// TwinCAT 3 PLC project DemoPLC
// ProgramVersion: 3.1.4026.22
// libraries:
//   Tc2_MC2, * (Beckhoff Automation GmbH)
//   Tc2_MDP, * (Beckhoff Automation GmbH)
//   Tc2_Standard, * (Beckhoff Automation GmbH)
//   Tc2_System, * (Beckhoff Automation GmbH)
//   Tc2_Utilities, * (Beckhoff Automation GmbH)
//   Tc3_IPCDiag, * (Beckhoff Automation GmbH)
// project tree:
//   DUTs/Bleutooth/ ST_Bleutooth.TcDUT, ST_BleutoothControl.TcDUT, ST_Bleutooth_Status.TcDUT
//   DUTs/CPU/ ST_CPUData.TcDUT, ST_CPUTemperature.TcDUT, ST_CPUUsage.TcDUT, ST_TaskData.TcDUT
//   DUTs/EtherCATJunction/ ST_MS4208_ETCOut.TcDUT
//   DUTs/General/ ST_EFU_Data.TcDUT, ST_EFU_Device_Inputs.TcDUT, ST_EFU_Inputs.TcDUT, ST_EFU_Outputs.TcDUT
//   DUTs/IO/DCombi/ ST_MO2338_DCombi.TcDUT
//   DUTs/IO/DI/ ST_DIS_Chanel_Diagnosis.TcDUT, ST_DIS_Diagnosis.TcDUT, ST_DIS_Inputs.TcDUT, ST_MO1008_DI.TcDUT
//   DUTs/IO/DO/ ST_DOS_Diagnosis.TcDUT, ST_DOS_Output.TcDUT, ST_DOS_Chanel_Diagnosis.TcDUT, ST_MO2008_DO.TcDUT
//   DUTs/PSU/ ST_PSU_Data.TcDUT, ST_PSU_Inputs.TcDUT, ST_PSU_Outputs.TcDUT
//   GVLs/ Global_Managed_Variables.TcGVL
//   / PlcTask.TcTTO
//   POUs/ FB_CollectCPUData.TcPOU, MAIN.TcPOU
//   POUs/Motion/Duts/ E_DemoSteps.TcTLEO, ST_PositionParameters.TcDUT
//   POUs/Motion/ FB_DemoMotion.TcPOU
//   POUs/Utilities/ FB_Blink.TcPOU
// real-time tasks:
//   TASK PlcTask: cycle T#10ms, priority 20, ADS port 350
// motion (NC):
//   TASK NC-Task 1 SAF: cycle T#2ms, priority 4, ADS port 501
//   TASK NC-Task 1 SVB: cycle T#10ms, priority 8, ADS port 511
//   AXIS Axis 2 (id 2)
//     General: UnitName=°
//     Dynamic: Acceleration=15000, Deceleration=15000, Jerk=118292.94
//     Velo: RefSearch=262.8732, RefSync=262.8732, SlowManual=1314.366, FastManual=7886.196, Fast=26287.32, Maximum=26287.32
//     OtherSettings: AllowMotionCmdToSlave=true
//     encoder EncType=19
//       EncPara: ScaleFactorNumerator=360, ScaleFactorDenominator=1048576, MaxCount=#xffffffff
//     drive DrvType=16
//       DrvPara: MaxCount=#xffffffff, DriveControlDWord=#x00020100
//         Analog: VeloReferenz=28916.052, VeloScale=32, TorqueSetpointScale=10, ScaleFactorActTorque=0.1
//         TimeComp: TaskDelayCycles=1
//     controller CtrType=1
//       CtrPara: PriorControlFactor=1
//         PID: PosKp=5
//         Observer: BandWidth=20
// I/O:
//   DEVICE Device 1 (EtherCAT), AmsNetId 10.201.45.9.2.1
//     Term 14 (MB1200-0000)
// variable links:
//   (this object) <-> Device 1 (EtherCAT)/Term 14 (MB1200-0000)/Term 8 (MB1100-0002)/Term 11 (MO7221-9016-1114)
//     Drive/Inputs/In/nDataIn1 <-> DRV Following error actual value/Following error actual value
//     Drive/Inputs/In/nDataIn3[0] <-> DRV Torque actual value/Torque actual value
//     Drive/Inputs/In/nDcOutputTime <-> InfoData/DcOutputShift
//     Drive/Inputs/In/nState1 <-> DRV Statusword/Statusword
//     Drive/Inputs/In/nState2 <-> DRV Statusword/Statusword @bit 8
//     Drive/Inputs/In/nState4 @bit 1 <-> WcState/InputToggle0
//     Drive/Inputs/In/nState4 <-> WcState/WcState0
//     Drive/Outputs/Out/nCtrl1 <-> DRV Controlword/Controlword
//     Drive/Outputs/Out/nCtrl2 <-> DRV Controlword/Controlword @bit 8
//     Drive/Outputs/Out/nDataOut1 <-> DRV Target position/Target position
//     Enc/Inputs/In/nDataIn1 <-> FB Position/Position
//     Enc/Inputs/In/nDcInputTime <-> InfoData/DcInputShift
//     Enc/Inputs/In/nState2 @bit 6 <-> FB Status/Status/Input cycle counter
//     Enc/Inputs/In/nState2 @bit 5 <-> FB Status/Status/TxPDO State
//     Enc/Inputs/In/nState4 @bit 1 <-> WcState/InputToggle0
//     Enc/Inputs/In/nState4 <-> WcState/WcState0
//     PlcTask Inputs/MAIN.fbDemoMotion.bSafety_Error <-> Module 1 (SafetyMDSingle)/Standard Inputdata/Standard Out Var 9
//     PlcTask Inputs/MAIN.fbDemoMotion.bSafety_OK <-> Module 1 (SafetyMDSingle)/Standard Inputdata/Standard Out Var 8
//     PlcTask Outputs/MAIN.bRunSafety <-> Module 1 (SafetyMDSingle)/Standard Outputdata/Standard In Var 2
//     PlcTask Outputs/MAIN.fbDemoMotion.bSafety_ErrorAckFromPLC <-> Module 1 (SafetyMDSingle)/Standard Outputdata/Standard In Var 1
//     PlcTask Outputs/MAIN.fbDemoMotion.bSafety_ErrorAckFromPLC <-> Module 1 (SafetyMDSingle)/Standard Outputdata/Standard In Var 7
//     PlcTask Outputs/MAIN.fbDemoMotion.bSafety_STOFromPLC <-> Module 1 (SafetyMDSingle)/Standard Outputdata/Standard In Var 6
//   (this object) <-> Device 1 (EtherCAT)/Term 14 (MB1200-0000)/Term 8 (MB1100-0002)
//     PlcTask Inputs/MAIN.stBleuToothData.Status/BleutoothEnabled <-> BTG Inputs/Status/Bluetooth Enabled
//     PlcTask Inputs/MAIN.stBleuToothData.Status/Connected <-> BTG Inputs/Status/Connected
//     PlcTask Inputs/MAIN.stBleuToothData.Status/Diag <-> BTG Inputs/Status/Diag
//     PlcTask Inputs/MAIN.stBleuToothData.Status/DonglePresent <-> BTG Inputs/Status/Dongle Present
//     PlcTask Inputs/MAIN.stBleuToothData.Status/Pairing <-> BTG Inputs/Status/Pairing Active
//     PlcTask Outputs/MAIN.stBleuToothData.control/ActivatePairingMode <-> BTG Outputs/Control/Activate Pairing
//     PlcTask Outputs/MAIN.stBleuToothData.control/EnableBleutoothDiagnosis <-> BTG Outputs/Control/Enable Bluetooth
//   (this object) <-> Device 1 (EtherCAT)/Term 14 (MB1200-0000)/Term 8 (MB1100-0002)/Term 16 (MS1010-1002-1334)
//     PlcTask Inputs/MAIN.stPSUData.stPSUInputs/DCOk <-> PSU Inputs/DC OK
//     PlcTask Inputs/MAIN.stPSUData.stPSUInputs/Overrange <-> PSU Inputs/Overrange
//     PlcTask Inputs/MAIN.stPSUData.stPSUInputs/bError <-> PSU Inputs/Error
//     PlcTask Inputs/MAIN.stPSUData.stPSUInputs/bI2TWarning <-> PSU Inputs/I2T Warning
//     PlcTask Inputs/MAIN.stPSUData.stPSUInputs/bWarning <-> PSU Inputs/Warning
//     PlcTask Inputs/MAIN.stPSUData.stPSUInputs/fActualOutputCurrent <-> PSU Inputs/Output Current
//     PlcTask Inputs/MAIN.stPSUData.stPSUInputs/fActualOutputVoltage <-> PSU Inputs/Output Voltage
//     PlcTask Inputs/MAIN.stPSUData.stPSUInputs/nActualI2TUtilization <-> PSU Inputs/I2T Utilization
//     PlcTask Inputs/MAIN.stPSUData.stPSUInputs/nInfoData1 <-> PSU Inputs/Info Data 1
//     PlcTask Inputs/MAIN.stPSUData.stPSUInputs/nInfoData2 <-> PSU Inputs/Info Data 2
//     PlcTask Outputs/MAIN.stPSUData.stPSUOutputs/bDisableOutput <-> PSU Outputs/Disable Output
//     PlcTask Outputs/MAIN.stPSUData.stPSUOutputs/bReset <-> PSU Outputs/Reset
//   (this object) <-> Device 1 (EtherCAT)/Term 14 (MB1200-0000)/Term 8 (MB1100-0002)/Term 18 (MB1120)/Term 19 (MS4208-2003-1112)
//     PlcTask Inputs/MAIN.st_MS4208_EtherCATOut.stEFUInputsDevice/bDiag <-> EFU Device Inputs/Diag
//     PlcTask Inputs/MAIN.st_MS4208_EtherCATOut.stEFUInputsDevice/bError <-> EFU Device Inputs/Error
//     PlcTask Inputs/MAIN.st_MS4208_EtherCATOut.stEFUInputsDevice/bOvertemperatureWarning <-> EFU Device Inputs/Overtemperature Warning
//     PlcTask Inputs/MAIN.st_MS4208_EtherCATOut.stEFUInputsDevice/bUnderVoltage_Up <-> EFU Device Inputs/Undervoltage Up
//     PlcTask Inputs/MAIN.st_MS4208_EtherCATOut.stEFUInputsDevice/bUnderVoltage_Us <-> EFU Device Inputs/Undervoltage Us
//     PlcTask Inputs/MAIN.st_MS4208_EtherCATOut.stEFUInputsDevice/bWarning <-> EFU Device Inputs/Warning
//     PlcTask Inputs/MAIN.st_MS4208_EtherCATOut.stEFUInputsDevice/fTotalCurrent <-> EFU Device Inputs/Total Current
//     PlcTask Inputs/MAIN.st_MS4208_EtherCATOut.stEFUUs.EFUInputs/bEnabled <-> EFU Us Inputs/Enabled
//     PlcTask Inputs/MAIN.st_MS4208_EtherCATOut.stEFUUs.EFUInputs/bError <-> EFU Us Inputs/Error
//     PlcTask Inputs/MAIN.st_MS4208_EtherCATOut.stEFUUs.EFUInputs/bTripped <-> EFU Us Inputs/Tripped
//     PlcTask Inputs/MAIN.st_MS4208_EtherCATOut.stEFUUs.EFUInputs/bWarning <-> EFU Us Inputs/Warning
//     PlcTask Inputs/MAIN.st_MS4208_EtherCATOut.stEFUUs.EFUInputs/fCurrent <-> EFU Us Inputs/Current
//     PlcTask Inputs/MAIN.st_MS4208_EtherCATOut.stEFU_Up1.EFUInputs/bEnabled <-> EFU Up1 Inputs/Enabled
//     PlcTask Inputs/MAIN.st_MS4208_EtherCATOut.stEFU_Up2.EFUInputs/bEnabled <-> EFU Up2 Inputs/Enabled
//     PlcTask Inputs/MAIN.st_MS4208_EtherCATOut.stEFU_Up1.EFUInputs/bError <-> EFU Up1 Inputs/Error
//     PlcTask Inputs/MAIN.st_MS4208_EtherCATOut.stEFU_Up2.EFUInputs/bError <-> EFU Up2 Inputs/Error
//     PlcTask Inputs/MAIN.st_MS4208_EtherCATOut.stEFU_Up1.EFUInputs/bTripped <-> EFU Up1 Inputs/Tripped
//     PlcTask Inputs/MAIN.st_MS4208_EtherCATOut.stEFU_Up2.EFUInputs/bTripped <-> EFU Up2 Inputs/Tripped
//     PlcTask Inputs/MAIN.st_MS4208_EtherCATOut.stEFU_Up1.EFUInputs/bWarning <-> EFU Up1 Inputs/Warning
//     PlcTask Inputs/MAIN.st_MS4208_EtherCATOut.stEFU_Up2.EFUInputs/bWarning <-> EFU Up2 Inputs/Warning
//     PlcTask Inputs/MAIN.st_MS4208_EtherCATOut.stEFU_Up1.EFUInputs/fCurrent <-> EFU Up1 Inputs/Current
//     PlcTask Inputs/MAIN.st_MS4208_EtherCATOut.stEFU_Up2.EFUInputs/fCurrent <-> EFU Up2 Inputs/Current
//     PlcTask Outputs/MAIN.st_MS4208_EtherCATOut.stEFUUs.EFUOutputs/ControlViaProcessData <-> EFU Us Outputs/Control via Process Data
//     PlcTask Outputs/MAIN.st_MS4208_EtherCATOut.stEFUUs.EFUOutputs/bEnable <-> EFU Us Outputs/Enable
//     PlcTask Outputs/MAIN.st_MS4208_EtherCATOut.stEFUUs.EFUOutputs/bReset <-> EFU Us Outputs/Reset
//     PlcTask Outputs/MAIN.st_MS4208_EtherCATOut.stEFU_Up1.EFUOutputs/ControlViaProcessData <-> EFU Up1 Outputs/Control via Process Data
//     PlcTask Outputs/MAIN.st_MS4208_EtherCATOut.stEFU_Up2.EFUOutputs/ControlViaProcessData <-> EFU Up2 Outputs/Control via Process Data
//     PlcTask Outputs/MAIN.st_MS4208_EtherCATOut.stEFU_Up1.EFUOutputs/bEnable <-> EFU Up1 Outputs/Enable
//     PlcTask Outputs/MAIN.st_MS4208_EtherCATOut.stEFU_Up2.EFUOutputs/bEnable <-> EFU Up2 Outputs/Enable
//     PlcTask Outputs/MAIN.st_MS4208_EtherCATOut.stEFU_Up1.EFUOutputs/bReset <-> EFU Up1 Outputs/Reset
//     PlcTask Outputs/MAIN.st_MS4208_EtherCATOut.stEFU_Up2.EFUOutputs/bReset <-> EFU Up2 Outputs/Reset
//   (this object) <-> Device 1 (EtherCAT)/Term 14 (MB1200-0000)/Term 8 (MB1100-0002)/Term 20 (MO1008-0000-1111)
//     PlcTask Inputs/MAIN.St_MO1008_DIData.EFUInputs/bEnabled <-> EFU Inputs/Enabled
//     PlcTask Inputs/MAIN.St_MO1008_DIData.EFUInputs/bError <-> EFU Inputs/Error
//     PlcTask Inputs/MAIN.St_MO1008_DIData.EFUInputs/bTripped <-> EFU Inputs/Tripped
//     PlcTask Inputs/MAIN.St_MO1008_DIData.EFUInputs/bWarning <-> EFU Inputs/Warning
//     PlcTask Inputs/MAIN.St_MO1008_DIData.EFUInputs/fCurrent <-> EFU Inputs/Current
//     PlcTask Outputs/MAIN.St_MO1008_DIData.ModuleDiagnostics.EFUOutputs/ControlViaProcessData <-> EFU Outputs/Control Via Process Data
//     PlcTask Outputs/MAIN.St_MO1008_DIData.ModuleDiagnostics.EFUOutputs/bEnable <-> EFU Outputs/Enable
//     PlcTask Outputs/MAIN.St_MO1008_DIData.ModuleDiagnostics.EFUOutputs/bReset <-> EFU Outputs/Reset
//   (this object) <-> Device 1 (EtherCAT)/Term 14 (MB1200-0000)/Term 8 (MB1100-0002)/Term 23 (MO2008-0000-1111)
//     PlcTask Inputs/MAIN.st_MO2008_DOData.EFUInputs/bEnabled <-> EFU Inputs/Enabled
//     PlcTask Inputs/MAIN.st_MO2008_DOData.EFUInputs/bError <-> EFU Inputs/Error
//     PlcTask Inputs/MAIN.st_MO2008_DOData.EFUInputs/bTripped <-> EFU Inputs/Tripped
//     PlcTask Inputs/MAIN.st_MO2008_DOData.EFUInputs/bWarning <-> EFU Inputs/Warning
//     PlcTask Inputs/MAIN.st_MO2008_DOData.ModuleDiagnostics.EFUInputs/fCurrent <-> EFU Inputs/Current
//     PlcTask Inputs/MAIN.st_MO2008_DOData.OutputDiagnostics/Chanel_0/PowersupplyMissing <-> DOS Diagnosis/Power Supply Missing
//     PlcTask Inputs/MAIN.st_MO2008_DOData.OutputDiagnostics/Chanel_0/bOpenLoad <-> DOS Diagnosis/Open Load
//     PlcTask Inputs/MAIN.st_MO2008_DOData.OutputDiagnostics/Chanel_0/bOvercurrent <-> DOS Diagnosis/Overcurrent
//     PlcTask Inputs/MAIN.st_MO2008_DOData.OutputDiagnostics/Chanel_0/bOverload <-> DOS Diagnosis/Overload
//     PlcTask Inputs/MAIN.st_MO2008_DOData.OutputDiagnostics/Chanel_0/bShortTo24V <-> DOS Diagnosis/Short to 24V
//     PlcTask Inputs/MAIN.st_MO2008_DOData.OutputDiagnostics/Chanel_{1..7}/PowersupplyMissing <-> DOS Diagnosis/Power Supply Missing_{1..7}  (7 links)
//     PlcTask Inputs/MAIN.st_MO2008_DOData.OutputDiagnostics/Chanel_{1..7}/bOpenLoad <-> DOS Diagnosis/Open Load_{1..7}  (7 links)
//     PlcTask Inputs/MAIN.st_MO2008_DOData.OutputDiagnostics/Chanel_{1..7}/bOvercurrent <-> DOS Diagnosis/Overcurrent_{1..7}  (7 links)
//     PlcTask Inputs/MAIN.st_MO2008_DOData.OutputDiagnostics/Chanel_{1..7}/bOverload <-> DOS Diagnosis/Overload_{1..7}  (7 links)
//     PlcTask Inputs/MAIN.st_MO2008_DOData.OutputDiagnostics/Chanel_{1..7}/bShortTo24V <-> DOS Diagnosis/Short to 24V_{1..7}  (7 links)
//     PlcTask Outputs/MAIN.st_MO2008_DOData.ModuleDiagnostics.EFUOutputs/ControlViaProcessData <-> EFU Outputs/Control Via Process Data
//     PlcTask Outputs/MAIN.st_MO2008_DOData.ModuleDiagnostics.EFUOutputs/bEnable <-> EFU Outputs/Enable
//     PlcTask Outputs/MAIN.st_MO2008_DOData.ModuleDiagnostics.EFUOutputs/bReset <-> EFU Outputs/Reset
//     PlcTask Outputs/MAIN.st_MO2008_DOData.OutputStatus/bOutputCh1 <-> DOS Output/Output
//     PlcTask Outputs/MAIN.st_MO2008_DOData.OutputStatus/bOutputCh{2..8} <-> DOS Output/Output_{1..7}  (7 links)
//   (this object) <-> Device 1 (EtherCAT)/Term 14 (MB1200-0000)/Term 8 (MB1100-0002)/Term 24 (MO2338-0000-1112)
//     PlcTask Inputs/MAIN.STD_MO2338_CombiData.DIDiagnostics/Chanel_0/bWirebreak <-> DIP Diagnosis/Wirebreak
//     PlcTask Inputs/MAIN.STD_MO2338_CombiData.DIDiagnostics/Chanel_{1..7}/bWirebreak <-> DIP Diagnosis/Wirebreak_{1..7}  (7 links)
//     PlcTask Inputs/MAIN.STD_MO2338_CombiData.DODisgnostics/Chanel_0/bOvercurrent <-> DOS Diagnosis/Overcurrent
//     PlcTask Inputs/MAIN.STD_MO2338_CombiData.DODisgnostics/Chanel_0/bOverload <-> DOS Diagnosis/Overload
//     PlcTask Inputs/MAIN.STD_MO2338_CombiData.DODisgnostics/Chanel_0/bShortTo24V <-> DOS Diagnosis/Short to 24V
//     PlcTask Inputs/MAIN.STD_MO2338_CombiData.DODisgnostics/Chanel_{1..7}/bOvercurrent <-> DOS Diagnosis/Overcurrent_{1..7}  (7 links)
//     PlcTask Inputs/MAIN.STD_MO2338_CombiData.DODisgnostics/Chanel_{1..7}/bOverload <-> DOS Diagnosis/Overload_{1..7}  (7 links)
//     PlcTask Inputs/MAIN.STD_MO2338_CombiData.DODisgnostics/Chanel_{1..7}/bShortTo24V <-> DOS Diagnosis/Short to 24V_{1..7}  (7 links)
//     PlcTask Inputs/MAIN.STD_MO2338_CombiData.EFUInputs/bError <-> DEV Inputs Device/Diag
//     PlcTask Inputs/MAIN.STD_MO2338_CombiData.EFUInputs/bWarning <-> DEV Inputs Device/Overtemperature
//     PlcTask Inputs/MAIN.STD_MO2338_CombiData.EFUInputs/fCurrent <-> EFU Inputs/Current
//     PlcTask Inputs/MAIN.STD_MO2338_CombiData.InputStatus/bInputCh1 <-> DIP Input/Input
//     PlcTask Inputs/MAIN.STD_MO2338_CombiData.InputStatus/bInputCh{2..8} <-> DIP Input/Input_{1..7}  (7 links)
//     PlcTask Inputs/MAIN.STD_MO2338_CombiData.ModuleDiagnostics/EFUInputs/bEnabled <-> EFU Inputs/Enabled
//     PlcTask Inputs/MAIN.STD_MO2338_CombiData.ModuleDiagnostics/EFUInputs/bError <-> EFU Inputs/Error
//     PlcTask Inputs/MAIN.STD_MO2338_CombiData.ModuleDiagnostics/EFUInputs/bTripped <-> EFU Inputs/Tripped
//     PlcTask Inputs/MAIN.STD_MO2338_CombiData.ModuleDiagnostics/EFUInputs/bWarning <-> EFU Inputs/Warning
//     PlcTask Outputs/MAIN.STD_MO2338_CombiData.OutputStatus/bOutputCh1 <-> EFU Outputs/Output
//     PlcTask Outputs/MAIN.STD_MO2338_CombiData.OutputStatus/bOutputCh{2..8} <-> EFU Outputs/Output_{1..7}  (7 links)
//   (this object) <-> NC-Task 1 SAF/Axes/Axis 2
//     PlcTask Inputs/MAIN.fbDemoMotion.ServoAxis.NcToPlc <-> Outputs/ToPlc
//     PlcTask Outputs/MAIN.fbDemoMotion.ServoAxis.PlcToNc <-> Inputs/FromPlc

CONFIGURATION DemoPLC
    RESOURCE PLC ON TwinCAT3
        TASK PlcTask(INTERVAL := T#10ms, PRIORITY := 20);
        PROGRAM MAIN WITH PlcTask : MAIN;
    END_RESOURCE
END_CONFIGURATION

// ---- DUTs/Bleutooth/ST_Bleutooth.TcDUT
TYPE ST_Bleutooth :
STRUCT
	Status AT%I*	: ST_Bleutooth_Status	; // status inputs
	control AT%Q*	: ST_BleutoothControl	; // Control Outputs
END_STRUCT
END_TYPE

// ---- DUTs/Bleutooth/ST_BleutoothControl.TcDUT
TYPE ST_BleutoothControl :
STRUCT
	EnableBleutoothDiagnosis	: BOOL;
	ActivatePairingMode			: BOOL;
END_STRUCT
END_TYPE

// ---- DUTs/Bleutooth/ST_Bleutooth_Status.TcDUT
TYPE ST_Bleutooth_Status :
STRUCT
	DonglePresent 		: BIT;
	BleutoothEnabled	: BIT;
	Pairing				: BIT;
	Connected			: BIT;
	Diag				: BIT;
	InputCycleCounter	: BIT; 			
END_STRUCT
END_TYPE

// ---- DUTs/CPU/ST_CPUData.TcDUT
TYPE ST_CPUData :
STRUCT
	stTemperatureData 	: ST_CPUTemperature	;
	stUsageData			: ST_CPUUsage		;
END_STRUCT
END_TYPE

// ---- DUTs/CPU/ST_CPUTemperature.TcDUT
TYPE ST_CPUTemperature :
STRUCT
	// temperature
	nCPUCurrentTemparature	: INT ; // The current temperature [°C] of the CPU core.
	nCPUMaximumTemperature	: INT ; // The maximum temperature [°C] of the CPU core that has been observed since the TwinCAT XAR start.
	nCPUTemperatureLimit	: INT	:= 70 ; // The temperature limit [°C] of the CPU core. Exceeding this limit leads to frequency throttling of the core.
	bInThermalThrottling	: BOOL	; // Is TRUE if one of the real-time cores is currently throttling its frequency due to the temperature limits being exceeded.
END_STRUCT
END_TYPE

// ---- DUTs/CPU/ST_CPUUsage.TcDUT
TYPE ST_CPUUsage :
STRUCT
	nCPUUsage			: UINT 	; // CPU usage (%)
	nMaxCPUUsage		: UINT	; // maximum cpu usage measured since last powerup
	nLimitCPUUsage		: UINT	:= 80; // Critical level for CPU usage
	nCPUOverload		: BOOL	; // CPU maximum use exceeded 
END_STRUCT
END_TYPE

// ---- DUTs/CPU/ST_TaskData.TcDUT
TYPE ST_TaskData :
STRUCT
	CycleTime 		: LREAL;
	LastExecTime	: LREAL;
	SystemLatency	: LREAL; 
END_STRUCT
END_TYPE

// ---- DUTs/EtherCATJunction/ST_MS4208_ETCOut.TcDUT
TYPE ST_MS4208_ETCOut :
STRUCT
	stEFUInputsDevice	AT%I* :	ST_EFU_Device_Inputs;	
	stEFUUs				:	ST_EFU_Data	;
	stEFU_Up1			:	ST_EFU_Data	;
	stEFU_Up2			:	ST_EFU_Data	;
END_STRUCT
END_TYPE

// ---- DUTs/General/ST_EFU_Data.TcDUT
TYPE ST_EFU_Data :
STRUCT
	EFUInputs 	AT%I*	: ST_EFU_Inputs	;
	EFUOutputs 	AT%Q*	: ST_EFU_Outputs;
END_STRUCT
END_TYPE

// ---- DUTs/General/ST_EFU_Device_Inputs.TcDUT
TYPE ST_EFU_Device_Inputs :
STRUCT
	bError					: BOOL ;
	bWarning				: BOOL ;
	bUnderVoltage_Us		: BOOL ;
	bUnderVoltage_Up		: BOOL ;
	bOvertemperatureWarning	: BOOL ;
	bDiag					: BOOL ;
	fTotalCurrent			: REAL ;
END_STRUCT
END_TYPE

// ---- DUTs/General/ST_EFU_Inputs.TcDUT
TYPE ST_EFU_Inputs :
STRUCT
	bWarning 	: BOOL;
	bError 		: BOOL;
	bTripped 	: BOOL;
	bEnabled 	: BOOL;
	//InputCycleCounter : BYTE;
	fCurrent 	: REAL;
END_STRUCT
END_TYPE

// ---- DUTs/General/ST_EFU_Outputs.TcDUT
TYPE ST_EFU_Outputs :
STRUCT
	bEnable 				: BOOL;
	ControlViaProcessData 	: BOOL;
	bReset 					: BOOL;
END_STRUCT
END_TYPE

// ---- DUTs/IO/DCombi/ST_MO2338_DCombi.TcDUT
TYPE ST_MO2338_DCombi EXTENDS ST_EFU_Data :
STRUCT
	InputStatus 		AT%I* : ST_DIS_Inputs		;
	DIDiagnostics		AT%I* : ST_DIS_Diagnosis	;
	
	OutputStatus		AT%Q* : ST_DOS_Output		;
	DODisgnostics		AT%I* : ST_DOS_Diagnosis	;	

	ModuleDiagnostics	AT%I*	: ST_EFU_Data		; 
END_STRUCT
END_TYPE

// ---- DUTs/IO/DI/ST_DIS_Chanel_Diagnosis.TcDUT
TYPE ST_DIS_Chanel_Diagnosis :
STRUCT
	bWirebreak 				: BOOL;
	bPowerSupplymissing	: BOOL;
END_STRUCT
END_TYPE

// ---- DUTs/IO/DI/ST_DIS_Diagnosis.TcDUT
TYPE ST_DIS_Diagnosis :
STRUCT
	Chanel_0	: ST_DIS_Chanel_Diagnosis ;
	Chanel_1	: ST_DIS_Chanel_Diagnosis ;
	Chanel_2	: ST_DIS_Chanel_Diagnosis ;
	Chanel_3	: ST_DIS_Chanel_Diagnosis ;
	Chanel_4	: ST_DIS_Chanel_Diagnosis ;
	Chanel_5	: ST_DIS_Chanel_Diagnosis ;
	Chanel_6	: ST_DIS_Chanel_Diagnosis ;
	Chanel_7	: ST_DIS_Chanel_Diagnosis ;
END_STRUCT
END_TYPE

// ---- DUTs/IO/DI/ST_DIS_Inputs.TcDUT
TYPE ST_DIS_Inputs :
STRUCT
	bInputCh1 : BOOL;
	bInputCh2 : BOOL;
	bInputCh3 : BOOL;
	bInputCh4 : BOOL;
	bInputCh5 : BOOL;
	bInputCh6 : BOOL;
	bInputCh7 : BOOL;
	bInputCh8 : BOOL;
END_STRUCT
END_TYPE

// ---- DUTs/IO/DI/ST_MO1008_DI.TcDUT
TYPE ST_MO1008_DI EXTENDS ST_EFU_Data :
STRUCT
	InputStatus			AT%I*	: ST_DIS_Inputs 	;
	InputDiagnostics	AT%I*	: ST_DIS_Diagnosis	;
	ModuleDiagnostics	: ST_EFU_Data		; 
END_STRUCT
END_TYPE

// ---- DUTs/IO/DO/ST_DOS_Diagnosis.TcDUT
TYPE ST_DOS_Diagnosis :
STRUCT
	Chanel_0	: ST_DOS_Chanel_Diagnosis;
	Chanel_1	: ST_DOS_Chanel_Diagnosis;
	Chanel_2	: ST_DOS_Chanel_Diagnosis;
	Chanel_3	: ST_DOS_Chanel_Diagnosis;
	Chanel_4	: ST_DOS_Chanel_Diagnosis;
	Chanel_5	: ST_DOS_Chanel_Diagnosis;
	Chanel_6	: ST_DOS_Chanel_Diagnosis;
	Chanel_7	: ST_DOS_Chanel_Diagnosis;
END_STRUCT
END_TYPE

// ---- DUTs/IO/DO/ST_DOS_Output.TcDUT
TYPE ST_DOS_Output :
STRUCT
	bOutputCh1	: BOOL;
	bOutputCh2	: BOOL;
	bOutputCh3	: BOOL;
	bOutputCh4	: BOOL;
	bOutputCh5	: BOOL;
	bOutputCh6	: BOOL;
	bOutputCh7	: BOOL;
	bOutputCh8	: BOOL;
END_STRUCT
END_TYPE

// ---- DUTs/IO/DO/ST_DOS_Chanel_Diagnosis.TcDUT
TYPE ST_DOS_Chanel_Diagnosis :
STRUCT
	bOvercurrent 		: BOOL;
	bOverload			: BOOL;
	bOpenLoad			: BOOL;
	bShortTo24V			: BOOL;
	PowersupplyMissing	: BOOL;
END_STRUCT
END_TYPE

// ---- DUTs/IO/DO/ST_MO2008_DO.TcDUT
TYPE ST_MO2008_DO EXTENDS ST_EFU_Data :
STRUCT
	OutputStatus		AT%Q*	: ST_DOS_Output		;
	OutputDiagnostics	AT%I*	: ST_DOS_Diagnosis	;
	ModuleDiagnostics	: ST_EFU_Data		; 
END_STRUCT
END_TYPE

// ---- DUTs/PSU/ST_PSU_Data.TcDUT
TYPE ST_PSU_Data :
STRUCT
	stPSUInputs		AT%I*	: ST_PSU_Inputs ;
	stPSUOutputs	AT%Q*	: ST_PSU_Outputs; 
END_STRUCT
END_TYPE

// ---- DUTs/PSU/ST_PSU_Inputs.TcDUT
TYPE ST_PSU_Inputs :
STRUCT
	bWarning 				: BOOL;
	bError 					: BOOL;
	bI2TWarning 			: BOOL;
	DCOk					: BOOL;
	Overrange				: BOOL;
	nInpuCycleCounter 		: UINT;
	fActualOutputVoltage 	: REAL;
	fActualOutputCurrent 	: REAL;
	nActualI2TUtilization 	: USINT;
	nInfoData1 				: UINT;
	nInfoData2 				: UINT;
END_STRUCT
END_TYPE

// ---- DUTs/PSU/ST_PSU_Outputs.TcDUT
TYPE ST_PSU_Outputs :
STRUCT
	bDisableOutput	: BOOL ;
	bReset			: BOOL ;
END_STRUCT
END_TYPE

// ---- POUs/Motion/Duts/E_DemoSteps.TcTLEO
{attribute 'qualified_only'}
{attribute 'strict'}
{attribute 'to_string'}
TYPE E_DemoSteps :
(
	Idle := 0,
	MoveToHomePos,
	WaitForhoming,
	CheckForManualCommand,
	ECGModeInit, // the goal is to display a ECG (ElectroCardioGram, or heartbeat signal)   
		ECG_P1,
		ECG_P2,
		ECG_PRSegment,
		ECG_Q,
		ECG_R,
		ECG_S1,
		ECG_S2,
		Ecg_STSegment,
		ECG_T1,
		ECG_T2,
		ECG_Idle,
		ECG_Finish,
	ManualModeInit,
	ManualMode,
	ManualIdle,
	Error
);
END_TYPE

// ---- POUs/Motion/Duts/ST_PositionParameters.TcDUT
TYPE ST_PositionParameters : // Full positioning command parameters
STRUCT
	fTargetPos		: LREAL;
	fVelocity		: LREAL;
	fAcceleration	: LREAL;
	fDeceleration	: LREAL; 
	fJerk			: LREAL;
	eBuffermode		: MC_BufferMode;
END_STRUCT
END_TYPE

// ---- GVLs/Global_Managed_Variables.TcGVL
{attribute 'qualified_only'}
VAR_GLOBAL
	Blink_Slow 	: BOOL	; // Slow blinking bit
	Blink_Fast	: BOOL	; // fast blinking Bit
	
END_VAR
VAR_GLOBAL CONSTANT
	ALWAYS_TRUE		: BOOL := TRUE	; // always true constant
	ALWAYS_FALSE	: BOOL := FALSE	; // ALways false constant 
END_VAR

// ---- POUs/MAIN.TcPOU
PROGRAM MAIN
VAR
// Power control
	bCmdPowerOff			: BOOL; // Power off command from HMI 
	tonPowerOff				: TON := (PT := T#3S); // Timer for power down
	bShuttingDown			: BOOL; // System is shutting down
	ntShutdown				: NT_Shutdown ;
	
// Bleutooth
	stBleuToothData			: ST_Bleutooth		;
	bEnableBleutooth		: BOOL	:= TRUE		;
//PSU
	stPSUData				: ST_PSU_Data		;
//EtherCAT
	st_MS4208_EtherCATOut	: ST_MS4208_ETCOut	;
// Digital IO
	St_MO1008_DIData		: ST_MO1008_DI		;
	st_MO2008_DOData		: ST_MO2008_DO		;
	STD_MO2338_CombiData	: ST_MO2338_DCombi	;
	
// Safety	
	bRunSafety	AT%Q*	: BOOL ; // Run Safet program

//CPU
	stCpuData				: ST_CPUData		; 
	stTaskData				: ST_TaskData		;
	fbCollectCPUData	: FB_CollectCPUData;

// Motion
	bCmdStartManualMotionControl	: BOOL; // manual motion control is active (false = DemoMode)
	bCmdStopDemoMotion				: BOOL; // Enable demo mode
	bDemoMotionActive				: BOOL; // Demo mode is active
	bManualMotionAcitve				: BOOL; // Manual motion control is active
	fbDemoMotion					: FB_DemoMotion;	

	
	
END_VAR
VAR //	GlobalFunctions 
	fbBlinkSlow	: FB_Blink;
	fbBlinkFast	: FB_Blink;
END_VAR

ExecGlobalFunctions();

//Enable bleutooth module
stBleuToothData.control.EnableBleutoothDiagnosis 	:= TRUE;
stBleuToothData.control.ActivatePairingMode			:= TRUE; //not stBleutooth.Status.Connected; 

bRunSafety := TRUE;

// Check for controlled shutdown command
ShutdownControl();

fbCollectCPUData();
stCpuData 	:= fbCollectCPUData.GetCPUData;
stTaskData 	:= fbCollectCPUData.GetTaskData;

// Demo motion control
fbDemoMotion.StopDemoMode 	:= bCmdStopDemoMotion;
fbDemoMotion.StartManualMode := bCmdStartManualMotionControl;

fbDemoMotion();

bManualMotionAcitve := fbDemoMotion.ManualModeActive;
bDemoMotionActive	:= fbDemoMotion.DemoModeActive;

METHOD ExecBleutoothControl
VAR_INPUT
END_VAR
END_METHOD

METHOD PROTECTED ExecGlobalFunctions // sets global menaged variables
fbBlinkSlow.TimeOff := 1000;
fbBlinkSlow.TimeOn 	:= 1000;
fbBlinkSlow();
Global_Managed_Variables.Blink_Slow := fbBlinkSlow.BlinkBit;
 
fbBlinkFast.TimeOff := 500;
fbBlinkFast.TimeOn 	:= 500;
fbBlinkFast();
Global_Managed_Variables.Blink_Fast := fbBlinkFast.BlinkBit;
END_METHOD

METHOD ShutdownControl // controlled shutdown of the MX system
VAR_INPUT
END_VAR

tonPowerOff(IN := bCmdPowerOff);

IF tonPowerOff.Q THEN 
	bCmdStopDemoMotion	:= TRUE;
	bShuttingDown		:= NOT bDemoMotionActive;
END_IF

ntShutdown(	START:= bShuttingDown, TMOUT:= T#5S);
END_METHOD

END_PROGRAM

// ---- POUs/FB_CollectCPUData.TcPOU
FUNCTION_BLOCK FB_CollectCPUData
VAR
	bFirstCycle				: BOOL := TRUE;	// First cycle of Function Call
	bExecuteRead 			: BOOL;
	tPeriod 				: TIME := T#500MS ;

	fbReadIPCTemperature 	: FB_IPCDiag_ReadParameterPeriodic 	;
	
	fbReadIPCUsage		 	: FB_IPCDiag_ReadParameterPeriodic 	;
	tInterval				: TIME := T#0.5S ; // Read interval
	
	
	stCPUData				: ST_CPUData ;
	fbDiagRegister			: FB_IPCDiag_Register ;
	
	stTaskData				: ST_TaskData;
	fbTcSyslatency			: TC_SysLatencyEx;
	
	arBuffer					: ARRAY [0..100] OF DINT ; 
	
	
END_VAR

// Initiate IPC diagnostics register
fbDiagRegister(bExecute := bFirstCycle);

IF fbDiagRegister.bValid THEN 
	bFirstCycle 	:= FALSE;
	bExecuteRead 	:= TRUE; 
END_IF

// Read and process data
mReadTemperatureData(); 
mReadCPUUsageData();

PROPERTY PUBLIC GetCPUData : ST_CPUData
GET
GetCPUData := stCPUData;
END_GET
END_PROPERTY

PROPERTY PUBLIC GetTaskData : ST_TaskData
GET
GetTaskData := stTaskData;
END_GET
END_PROPERTY

METHOD PRIVATE mReadCPUUsageData : ST_CPUUsage
VAR
	nCPUUsage				: UINT ; // current cPU usage [%] 
	TaskIndex		: DINT ; // current task index
END_VAR
// read temperature diagnostic data
fbReadIPCUsage(
	bEnable:= TRUE, 
	eParameterKey:= E_IPCDiag_ParameterKey.CPU_Usage, 
	tPeriod:= T#1S, 
	fbRegister:= fbDiagRegister );

fbTcSyslatency(bExecute := fbReadIPCUsage.bValid);
	
// Process data
IF fbReadIPCUsage.bValid THEN 
	fbReadIPCUsage.GetParameter(pBuffer := ADR(nCPUUsage), nBufferSize := SIZEOF(nCPUUsage)) ;
	stCPUData.stUsageData.nCPUUsage		:= nCPUUsage;
	stCPUData.stUsageData.nMaxCPUUsage 	:= MAX(nCPUUsage, stCPUData.stUsageData.nMaxCPUUsage);
	stCPUData.stUsageData.nCPUOverload	:= nCPUUsage > stCPUData.stUsageData.nLimitCPUUsage;

	TaskIndex := GETCURTASKINDEXEX();
	stTaskData.CycleTime	:= _TaskInfo[TaskIndex].CycleTime / 10000.0; //convert 100ns to ms
	stTaskData.LastExecTime	:= _TaskInfo[TaskIndex].LastExecTime / 10000.0; //convert 100ns to ms
	stTaskData.SystemLatency:= fbTcSyslatency.nActual;
END_IF
END_METHOD

METHOD PRIVATE mReadTemperatureData : ST_CPUTemperature 
VAR
	nCPUTemperature : INT ;
END_VAR
// read temperature diagnostic data
fbReadIPCTemperature(
	bEnable:= bExecuteRead, 
	eParameterKey:= E_IPCDiag_ParameterKey.CPU_Temp, 
	tPeriod:= T#1S, 
	fbRegister:= fbDiagRegister );
	
// Process data
IF fbReadIPCTemperature.bValid THEN 
	fbReadIPCTemperature.GetParameter(pBuffer := ADR(nCPUTemperature), nBufferSize := SIZEOF(nCPUTemperature)) ;
	stCPUData.stTemperatureData.nCPUCurrentTemparature	:= nCPUTemperature;
	stCPUData.stTemperatureData.nCPUMaximumTemperature	:= MAX(nCPUTemperature, stCPUData.stTemperatureData.nCPUMaximumTemperature);
	stCPUData.stTemperatureData.bInThermalThrottling 	:= nCPUTemperature >= stCPUData.stTemperatureData.nCPUTemperatureLimit;
END_IF
END_METHOD

END_FUNCTION_BLOCK

// ---- POUs/Motion/FB_DemoMotion.TcPOU
FUNCTION_BLOCK INTERNAL FB_DemoMotion
VAR_INPUT
END_VAR
VAR_OUTPUT
END_VAR
VAR
	fMAXVELOCITY		: LREAL := 26000;//12000; // maximum motor velocity
	fMaxAcceleration	: LREAL := 15000;// 302143; // Maximum Motor acceleration
	fMaxDeceleration	: LREAL := 15000;// 302143; // Maximum Motor acceleration
END_VAR
VAR
	// Organisational bits
	tonEnebleDelay		: TON := (PT := T#5S); // On delay time between STO release and Enable
	bCmdEnableMotion	: BOOL ; // command activate motion
	bMotionEnabled		: BOOL ; // motion is in enabled state
	fOverride			: LREAL	:= 100.0; // override factor (default = 100%)
	
	bSafety_Error					AT%I*	: BOOL ; // Safety has error
	bSafety_STOFromPLC				AT%Q*	: BOOL ; // Sto releaste from PLC
	bSafety_ErrorAckFromPLC			AT%Q*	: BOOL ; // Safety error acknowledge from PLC
	
//	bCmdStartDemo		: BOOL ; // command activate demo mode
	rtStopDemoMode		: R_TRIG	; // Trigger for toggeling demo mode stop
	bCmdStopDemoMode	: BOOL ; // command stop demo mode
	bDemoModeActive		: BOOL ; // Demo mode is active

	bCmdStartManualMode	: BOOL ; // command activate manual mode
	bManualModeActive	: BOOL ; // Manual mode is active
	tofManualTimeOut	: TOF := (PT := T#30S); // Timeout for manual commands, if no commands are given then demo mode will be reactivated 

	ServoAxis			: AXIS_REF ; // Main servo axis

	bSafety_OK	AT%I* 	: BOOL ; // Safety Ok 
	// DemoMode
	eDemoStep			: E_DemoSteps 	; // Motion demo stepper
	eLastErrorStep		: E_DemoSteps	; // Active step when error occured
	
	//Parameters
	fHomePos			: LREAL := 75; // Home position (offset)
	
	tPRSegmentLength	: TIME := T#300MS 	; // length of the pr segment
	tSTSegmentLength	: TIME := T#300MS 	; // length of the ST segment
	tBetweenHeartbeats	: TIME := T#1S	; // Time between hearbeats
	
	Par_ToHomePosition	: ST_PositionParameters :=(fTargetPos 	:= 0, 
												fVelocity 		:= fMAXVELOCITY, 
												fAcceleration 	:= fMaxAcceleration, 
												fDeceleration 	:= fMaxDeceleration, 
												fJerk 			:= 0,
												eBuffermode		:= MC_BufferMode.MC_Aborting);

	Par_ECGP1			: ST_PositionParameters :=(fTargetPos 	:= 30, 
												fVelocity 		:= fMAXVELOCITY / 4, 
												fAcceleration 	:= fMaxAcceleration / 10, 
												fDeceleration 	:= fMaxDeceleration / 30, 
												fJerk 			:= 0,
												eBuffermode		:= MC_BufferMode.MC_Buffered);

	Par_ECGP2			: ST_PositionParameters :=(fTargetPos 	:= 0, 
												fVelocity 		:= fMAXVELOCITY / 3, 
												fAcceleration 	:= fMaxAcceleration / 15,
												fDeceleration 	:= fMaxDeceleration / 10, 
												fJerk 			:= 0,
												eBuffermode		:= MC_BufferMode.MC_Buffered);

	Par_ECGQ			: ST_PositionParameters :=(fTargetPos 	:= -30, 
												fVelocity 		:= fMAXVELOCITY / 2, 
												fAcceleration 	:= fMaxAcceleration, 
												fDeceleration 	:= fMaxDeceleration, 
												fJerk 			:= 0,
												eBuffermode		:= MC_BufferMode.MC_Buffered);

	Par_ECGR			: ST_PositionParameters :=(fTargetPos 	:= 360, 
												fVelocity 		:= fMAXVELOCITY, 
												fAcceleration 	:= fMaxAcceleration, 
												fDeceleration 	:= fMaxDeceleration, 
												fJerk 			:= 0,
												eBuffermode		:= MC_BufferMode.MC_Buffered);

	Par_ECGS1			: ST_PositionParameters :=(fTargetPos 	:= -120, 
												fVelocity 		:= fMAXVELOCITY, 
												fAcceleration 	:= fMaxAcceleration, 
												fDeceleration 	:= fMaxDeceleration, 
												fJerk 			:= 0,
												eBuffermode		:= MC_BufferMode.MC_Buffered);
								
	Par_ECGS2			: ST_PositionParameters :=(fTargetPos 	:= 0, 
												fVelocity 		:= fMAXVELOCITY / 2, 
												fAcceleration 	:= fMaxAcceleration, 
												fDeceleration 	:= fMaxDeceleration, 
												fJerk 			:= 0,
												eBuffermode		:= MC_BufferMode.MC_Buffered);

	Par_ECGT1			: ST_PositionParameters :=(fTargetPos 	:= 50, 
												fVelocity 		:= fMAXVELOCITY / 4, 
												fAcceleration 	:= fMaxAcceleration / 10, 
												fDeceleration 	:= fMaxDeceleration / 30, 
												fJerk 			:= 0,
												eBuffermode		:= MC_BufferMode.MC_Buffered);

	Par_ECGT2			: ST_PositionParameters :=(fTargetPos 	:= 0, 
												fVelocity 		:= fMAXVELOCITY / 2, 
												fAcceleration 	:= fMaxAcceleration / 10, 
												fDeceleration 	:= fMaxDeceleration, 
												fJerk 			:= 0,
												eBuffermode		:= MC_BufferMode.MC_Buffered);
 
	// Axis organizational functions
	tonSegment 		: TON 		; // Timer between segments  
	fbMCPower 		: MC_Power 	;
	fbMCReset		: MC_Reset 	;

	// Axis demoe Motion functions
	stActiveStepCommandParameters	: ST_PositionParameters; // Paremeters forwarded by the (latest) Active step
	bCmdExecuteMove		: BOOL 				; // Execute move command (Automatically switches between FBMoveAbsolute instances for queing)
	reMoveAbsoluteActive: R_TRIG 			; // Triggers when one of the move Absolute functions becomes active 
	bMoveAbsoluteDone	: BOOL				; // Move absolute command is done 
	fbMCMoveAbsolute_1 		: MC_MoveAbsolute 	;
	fbMCMoveAbsolute_2 		: MC_MoveAbsolute 	;
END_VAR


OrganisationalFunctions();

RunDemo();

PROPERTY DemoModeActive : bool
GET
IF bCmdStopDemoMode AND bDemoModeActive THEN 
	DemoModeActive := Global_Managed_Variables.Blink_Slow;	
ELSIF bDemoModeActive THEN 
	DemoModeActive := TRUE;	
END_IF
END_GET
END_PROPERTY

PROPERTY PUBLIC ManualModeActive : Bool
GET
ManualModeActive := bManualModeActive;
END_GET
END_PROPERTY

METHOD INTERNAL OrganisationalFunctions : BOOL
VAR_INPUT
END_VAR
// Release STO when Safety i opperational

// For now, automatically reset the safety
IF bSafety_Error THEN 
	{warning 'add error message handling'}
	bSafety_STOFromPLC 		:= FALSE;
	bSafety_ErrorAckFromPLC := TRUE;
ELSE
	bSafety_STOFromPLC 		:= TRUE;
	bSafety_ErrorAckFromPLC := FALSE;
END_IF

tonEnebleDelay(IN := bCmdEnableMotion OR bSafety_OK);

fbMCPower(	Axis 			:= ServoAxis, 
			Enable			:= tonEnebleDelay.Q,
			Enable_Positive	:= TRUE,
			Enable_Negative	:= TRUE,
			Override		:= fOverride,
			Status			=> bMotionEnabled,
			Error			=>,
			ErrorID			=>);
			
fbMCReset(	Axis 	:= ServoAxis);

IF fbMCPower.Status THEN 
	ServoAxis.ReadStatus();
END_IF
END_METHOD

METHOD RunDemo : BOOL
VAR_INPUT
END_VAR
// Manual mode control

// The following stepper is designed to mimick an ECG scan (Heartbeat) when looking at the position graph
CASE eDemoStep OF
	E_DemoSteps.Idle:
		bDemoModeActive 	:= FALSE;		
		bManualModeActive 	:= FALSE;		
		IF bMotionEnabled THEN 
			eDemoStep := E_DemoSteps.CheckForManualCommand;
		END_IF
	E_DemoSteps.CheckForManualCommand:
		IF bCmdStartManualMode THEN 
			bDemoModeActive 	:= FALSE;
			bCmdStopDemoMode 	:= FALSE;
			eDemoStep := E_DemoSteps.ManualModeInit;
		ELSIF bCmdStopDemoMode THEN 
			bDemoModeActive := FALSE;// Stay idle and wait for further command
		ELSIF bDemoModeActive THEN 
			eDemoStep := E_DemoSteps.ECG_P1;
		ELSE
			eDemoStep := E_DemoSteps.MoveToHomePos;
		END_IF
	// this section is only used when swithcing from manual to demo mode
	E_DemoSteps.MoveToHomePos:
		stActiveStepCommandParameters := Par_ToHomePosition;
		IF reMoveAbsoluteActive.Q OR bMoveAbsoluteDone THEN // Wait until the command is executed then move to next step
			eDemoStep := E_DemoSteps.WaitForhoming;
		ELSIF ServoAxis.NcToPlc.ActPos > -0.5 AND ServoAxis.NcToPlc.ActPos < 0.5 THEN // Servo is already at home position
			eDemoStep := E_DemoSteps.ECGModeInit;
			bCmdExecuteMove := FALSE;					
		ELSE
			bCmdExecuteMove := TRUE;					
		END_IF
	E_DemoSteps.WaitForhoming:
		IF bMoveAbsoluteDone THEN 
			eDemoStep := E_DemoSteps.ECGModeInit;
		END_IF
	E_DemoSteps.ECGModeInit:
		IF NOT ServoAxis.Status.Error THEN 
			bDemoModeActive := TRUE;
			eDemoStep := E_DemoSteps.ECG_P1;
		ELSE 
			eLastErrorStep := eDemoStep;
			eDemoStep := E_DemoSteps.Error;
	END_IF
	// Demo mode Creates ECG image on position scope
	E_DemoSteps.ECG_P1:
		stActiveStepCommandParameters := Par_ECGP1;
		IF reMoveAbsoluteActive.Q THEN // Wait until the command is executed then move to next step
			eDemoStep := E_DemoSteps.ECG_P2;
		ELSE
			bCmdExecuteMove := TRUE;		
		END_IF
	E_DemoSteps.ECG_P2:
		stActiveStepCommandParameters := Par_ECGP2;
		IF reMoveAbsoluteActive.Q THEN
			eDemoStep := E_DemoSteps.ECG_PRSegment;
		ELSE
			bCmdExecuteMove := TRUE;		
		END_IF			
	E_DemoSteps.ECG_PRSegment:
		IF tonSegment.Q THEN
			tonSegment.IN := FALSE;
			eDemoStep := E_DemoSteps.ECG_Q;			
		ELSIF bMoveAbsoluteDone THEN 
			tonSegment.PT := tPRSegmentLength ; 
			tonSegment.IN := TRUE;
		END_IF
	E_DemoSteps.ECG_Q:
		stActiveStepCommandParameters := Par_ECGQ;
		IF reMoveAbsoluteActive.Q THEN
			eDemoStep := E_DemoSteps.ECG_R;
		ELSE
			bCmdExecuteMove := TRUE;		
		END_IF			
	E_DemoSteps.ECG_R:
		stActiveStepCommandParameters := Par_ECGR;
		IF reMoveAbsoluteActive.Q THEN
			eDemoStep := E_DemoSteps.ECG_S1;
		ELSE
			bCmdExecuteMove := TRUE;		
		END_IF			
	E_DemoSteps.ECG_S1:
		stActiveStepCommandParameters := Par_ECGS1;
		IF reMoveAbsoluteActive.q THEN
			eDemoStep := E_DemoSteps.ECG_S2;
		ELSE
			bCmdExecuteMove := TRUE;		
		END_IF			
	E_DemoSteps.ECG_S2:
		stActiveStepCommandParameters := Par_ECGS2;
		IF reMoveAbsoluteActive.q THEN
			eDemoStep := E_DemoSteps.Ecg_STSegment;
		ELSE
			bCmdExecuteMove := TRUE;		
		END_IF			
	E_DemoSteps.Ecg_STSegment:
		IF tonSegment.Q THEN
			tonSegment.IN := FALSE;
			eDemoStep := E_DemoSteps.ECG_T1;			
		ELSIF bMoveAbsoluteDone THEN 
			tonSegment.PT := tSTSegmentLength ; 
			tonSegment.IN := TRUE;
		END_IF
	E_DemoSteps.ECG_T1:
		stActiveStepCommandParameters := Par_ECGT1;
		IF reMoveAbsoluteActive.Q THEN 
			eDemoStep := E_DemoSteps.ECG_T2;
		ELSE
			bCmdExecuteMove := TRUE;		
		END_IF
	E_DemoSteps.ECG_T2:
		stActiveStepCommandParameters := Par_ECGT2;
		IF reMoveAbsoluteActive.Q THEN
			eDemoStep := E_DemoSteps.ECG_Idle;
		ELSE
			bCmdExecuteMove := TRUE;		
		END_IF			
	E_DemoSteps.ECG_Idle:
		IF tonSegment.Q THEN
			tonSegment.IN := FALSE;
			eDemoStep := E_DemoSteps.CheckForManualCommand;		// End of ECG cycle, Return	
		ELSIF bMoveAbsoluteDone THEN 
			tonSegment.PT :=  tBetweenHeartbeats; 
			tonSegment.IN := TRUE;
		END_IF
	// Manual control
	E_DemoSteps.ManualModeInit:
		IF NOT ServoAxis.Status.Error AND not ServoAxis.Status.HasJob THEN 
			bCmdStartManualMode := FALSE;
			bManualModeActive := TRUE;
			eDemoStep := E_DemoSteps.ManualMode;
		ELSIF ServoAxis.Status.Error THEN 
			eDemoStep := E_DemoSteps.Error;
			{warning 'error message needs to be added'}
		END_IF
	E_DemoSteps.ManualMode:
		tofManualTimeOut.in := TRUE;
		IF NOT ServoAxis.Status.HasJob THEN 
			eDemoStep := E_DemoSteps.ManualIdle;
		END_IF
	E_DemoSteps.ManualIdle:
		tofManualTimeOut.IN := FALSE;
		IF ServoAxis.Status.HasJob THEN 
			eDemoStep := E_DemoSteps.ManualMode;
		ELSIF NOT tofManualTimeOut.q THEN // If no manual command is given, return to home position in order to start ECG again
			bManualModeActive := FALSE;
			eDemoStep := E_DemoSteps.MoveToHomePos;
		ELSIF NOT bManualModeActive THEN
			eDemoStep := E_DemoSteps.MoveToHomePos;
		END_IF
	// Housekeeping
	E_DemoSteps.Error:
		{warning 'add error handling'}
		bCmdExecuteMove := FALSE;
		IF ServoAxis.Status.Error THEN 
			fbMCReset.Execute := TRUE;
		ELSE
			fbMCReset.Execute := FALSE;
			eDemoStep := E_DemoSteps.Idle;
		END_IF
END_CASE

tonSegment();
tofManualTimeOut();

// Execute move absolute functions
// Move absolute commands can be stacked ensuring quick transitions and easy coding
fbMCMoveAbsolute_1( Execute		:= NOT fbMCMoveAbsolute_1.Busy AND bCmdExecuteMove,	
					Axis 		:= ServoAxis,
					Position	:= fHomePos + stActiveStepCommandParameters.fTargetPos,
					Velocity	:= stActiveStepCommandParameters.fVelocity,
					Acceleration:= stActiveStepCommandParameters.fAcceleration,
					Deceleration:= stActiveStepCommandParameters.fDeceleration,
					Jerk		:= stActiveStepCommandParameters.fJerk,
					BufferMode	:= stActiveStepCommandParameters.eBuffermode
					);
fbMCMoveAbsolute_2( Execute		:= fbMCMoveAbsolute_1.Busy AND bCmdExecuteMove,
					Axis 		:= ServoAxis,
					Position	:= fHomePos + stActiveStepCommandParameters.fTargetPos,
					Velocity	:= stActiveStepCommandParameters.fVelocity,
					Acceleration:= stActiveStepCommandParameters.fAcceleration,
					Deceleration:= stActiveStepCommandParameters.fDeceleration,
					Jerk		:= stActiveStepCommandParameters.fJerk,
					BufferMode	:= stActiveStepCommandParameters.eBuffermode
					);

reMoveAbsoluteActive(CLK := fbMCMoveAbsolute_1.Active OR fbMCMoveAbsolute_2.Active);
bMoveAbsoluteDone	:= fbMCMoveAbsolute_1.Done OR fbMCMoveAbsolute_2.Done;

IF reMoveAbsoluteActive.Q THEN 
	bCmdExecuteMove := FALSE;
ELSIF fbMCMoveAbsolute_1.Error OR fbMCMoveAbsolute_2.Error THEN 
	eLastErrorStep := eDemoStep;
	eDemoStep := E_DemoSteps.Error;
END_IF

{warning 'error message needs to be added'}
END_METHOD

PROPERTY StartManualMode : Bool
SET
// only starts the Manual mode, Manaul mode will stop automatically after 30Sec of no commands
IF StartManualMode AND NOT bManualModeActive THEN
	bCmdStartManualMode := TRUE;
END_IF
END_SET
END_PROPERTY

PROPERTY StopDemoMode : Bool
SET
// Demo needs to finish it's cycle before switching off, therefore the StopDemo command is triggered to bring the demo cycle to a controlled end
rtStopDemoMode(CLK := StopDemoMode);
IF rtStopDemoMode.Q THEN
	IF bManualModeActive THEN // Then manual made is active, turn off Manual mode to resume demo mode
		bManualModeActive 	:= FALSE;
		bCmdStartManualMode	:= FALSE;
	ELSE
		bCmdStopDemoMode := NOT bCmdStopDemoMode;
	END_IF
END_IF
END_SET
END_PROPERTY

END_FUNCTION_BLOCK

// ---- POUs/Utilities/FB_Blink.TcPOU
FUNCTION_BLOCK FB_Blink // creates a blinking bit with variable on and off time (Default 500ms off 500ms on) 
VAR_INPUT
END_VAR
VAR_OUTPUT
END_VAR
VAR
	OnTimer		: TON := (PT := T#500MS); 
	OffTimer	: TON := (PT := T#500MS);
END_VAR

OnTimer	(IN := NOT OffTimer.Q);
OffTimer(IN := OnTimer.Q);

PROPERTY BlinkBit : Bool
GET
BlinkBit := OnTimer.Q;
END_GET
END_PROPERTY

PROPERTY TimeOff : Uint
SET
OffTimer.PT := UINT_TO_TIME(TimeOff);
END_SET
END_PROPERTY

PROPERTY TimeOn : UINT // Time on [MS]
SET
OnTimer.PT := UINT_TO_TIME(TimeOn);
END_SET
END_PROPERTY

END_FUNCTION_BLOCK
